// TIA Portal V20 export
TYPE "typeCmControlNodeBrakeTest"
// stored: Namespace Unit1.Em8
   STRUCT
      thicknessAxisZ : "LER_typeBrakeTestEmControlNodes";
   END_STRUCT;
END_TYPE
